// TIA Portal V18 export
PlcTagTable "Default tag table"
  PlcTag "HMI_Run_Enable"  LogicalAddress=%M20.0
  PlcTag "HMI_Reset_Alarm"  LogicalAddress=%M20.1
  PlcTag "HMI_Che_Do_Thi"  LogicalAddress=%M20.2
  PlcTag "HMI_Sim_Mode"  LogicalAddress=%M20.3
  PlcTag "PLC1_State"  LogicalAddress=%MW12
  PlcTag "PLC1_Loi_Tong"  LogicalAddress=%M20.4
  PlcTag "PLC1_Stop_Active"  LogicalAddress=%M20.5
  PlcTag "PLC1_EStop_Latch"  LogicalAddress=%M20.6
  PlcTag "PLC1_SP_Valid"  LogicalAddress=%M20.7
  PlcTag "Nut_Khoi_Dong_HMI"  LogicalAddress=%M21.0
  PlcTag "Nut_Dung_HMI"  LogicalAddress=%M21.1
  PlcTag "Nut_Reset_HMI"  LogicalAddress=%M21.2
  PlcTag "HMI_VFD_Bon2_Comm_Enable"  LogicalAddress=%M21.3
  PlcTag "HMI_VFD_Bon2_Real_Enable"  LogicalAddress=%M21.4
  PlcTag "HMI_PID_Bon2_Dau_Noi_Enable"  LogicalAddress=%M21.5
  PlcTag "PID_Bon2_Enable"  LogicalAddress=%M21.6
  PlcTag "PID_Bon2_Enable_Eff"  LogicalAddress=%M21.7
  PlcTag "PID_Bon2_SP"  LogicalAddress=%MD30
  PlcTag "PID_Bon2_PV_Eff"  LogicalAddress=%MD34
  PlcTag "PID_Bon2_CV"  LogicalAddress=%MD38
  PlcTag "HMI_SP_PLC1_Nhiet_Do_Bon2"  LogicalAddress=%MD42
  PlcTag "HMI_SP_PLC1_Toc_Do_Bon2_Main"  LogicalAddress=%MD46
  PlcTag "TT3208_Bon2_Eff"  LogicalAddress=%MD50
  PlcTag "TT3208_Bon2_HMI"  LogicalAddress=%MD54
  PlcTag "VFD_Bon2_Toc_Do_Cmd"  LogicalAddress=%MD58
  PlcTag "TT3208_Bon2_Use_HMI"  LogicalAddress=%M22.0
  PlcTag "VFD_Bon2_MB_Error"  LogicalAddress=%M22.1
  PlcTag "VFD_Bon2_MB_Busy"  LogicalAddress=%M22.2
  PlcTag "VFD_Bon2_MB_Done"  LogicalAddress=%M22.3
  PlcTag "MB_TCP_ERROR"  LogicalAddress=%M22.4
  PlcTag "MB_TCP_BUSY"  LogicalAddress=%M22.5
  PlcTag "MB_TCP_DONE"  LogicalAddress=%M22.6
  PlcTag "PLC1_Heartbeat_Timeout"  LogicalAddress=%M22.7
  PlcTag "VFD_Bon2_MB_ControlWord"  LogicalAddress=%MW62
  PlcTag "VFD_Bon2_MB_StatusWord"  LogicalAddress=%MW64
  PlcTag "VFD_Bon2_MB_FreqSetpoint"  LogicalAddress=%MW66
  PlcTag "VFD_Bon2_MB_FreqActual"  LogicalAddress=%MW68
  PlcTag "VFD_Bon2_MB_Status"  LogicalAddress=%MW70
  PlcTag "MB_TCP_STATUS"  LogicalAddress=%MW72
  PlcTag "MB_TCP_iStep"  LogicalAddress=%MW74
  PlcTag "PLC1_Heartbeat"  LogicalAddress=%MW76
  PlcTag "PLC2_Heartbeat_Recv"  LogicalAddress=%MW78
  PlcTag "VFD_Bon2_Contactor"  LogicalAddress=%Q0.0
  PlcTag "CV3201_Nuoc_Bon1_M"  LogicalAddress=%MD1200
  PlcTag "CV3206_Hoi_Bon2_M"  LogicalAddress=%MD1208
  PlcTag "CV3304_Nuoc_Lam_Mat_M"  LogicalAddress=%MD1232
  PlcTag "FQ3200_Bon1_Eff"  LogicalAddress=%MD712
  PlcTag "FQ3205_Bon2_Eff"  LogicalAddress=%MD744
  PlcTag "FT3309_Xa_Thanh_Pham_Eff"  LogicalAddress=%MD880
  PlcTag "HMI_Anim_Bon1_Frame"  LogicalAddress=%MW260
  PlcTag "HMI_Anim_Bon1_MucDich"  LogicalAddress=%MW262
  PlcTag "HMI_Anim_Bon2_Frame"  LogicalAddress=%MW264
  PlcTag "HMI_Anim_Bon2_MucDich"  LogicalAddress=%MW266
  PlcTag "HMI_Anim_BonChua1_MucDich"  LogicalAddress=%MW268
  PlcTag "HMI_Anim_BonChua2_MucDich"  LogicalAddress=%MW270
  PlcTag "LT3203_Bon1_Eff"  LogicalAddress=%MD720
  PlcTag "LT3209_Bon2_Eff"  LogicalAddress=%MD752
  PlcTag "LT3302_BonChua1_Eff"  LogicalAddress=%MD832
  PlcTag "LT3307_BonChua2_Eff"  LogicalAddress=%MD856
  PlcTag "PI3308_Truoc_Filter_Eff"  LogicalAddress=%MD872
  PlcTag "Pump3264_Chuyen_Nhanh1"  LogicalAddress=%M100.0
  PlcTag "Pump3265_Chuyen_Nhanh2"  LogicalAddress=%M100.1
  PlcTag "Pump3361_LuanChuyen_BonChua1"  LogicalAddress=%M100.2
  PlcTag "Pump3362_Xa_BonChua1"  LogicalAddress=%M100.3
  PlcTag "Pump3364_Filter"  LogicalAddress=%M100.4
  PlcTag "Pump3365_Filter"  LogicalAddress=%M100.5
  PlcTag "TT3204_Bon1_Eff"  LogicalAddress=%MD728
  PlcTag "TT3301_BonChua1_Eff"  LogicalAddress=%MD840
  PlcTag "TT3303_TraoDoiNhiet_Eff"  LogicalAddress=%MD848
  PlcTag "TT3306_BonChua2_Eff"  LogicalAddress=%MD864
  PlcTag "V3230_Nuoc_Bon1"  LogicalAddress=%M100.6
  PlcTag "V3232_Xa_Bon1"  LogicalAddress=%M100.7
  PlcTag "V3233_Xa_Bon1"  LogicalAddress=%M101.0
  PlcTag "V3234_Xa_Bon1"  LogicalAddress=%M101.1
  PlcTag "V3235_Nuoc_Bon2"  LogicalAddress=%M101.2
  PlcTag "V3237_Xa_Bon2"  LogicalAddress=%M101.3
  PlcTag "V3238_Xa_Bon2"  LogicalAddress=%M101.4
  PlcTag "V3239_Xa_Bon2"  LogicalAddress=%M101.5
  PlcTag "V3331_Xa_BonChua1"  LogicalAddress=%M101.6
  PlcTag "V3332_Xa_BonChua1"  LogicalAddress=%M101.7
  PlcTag "V3333_DieuHuong_BonChua1"  LogicalAddress=%M102.0
  PlcTag "V3334_DieuHuong_BonChua1"  LogicalAddress=%M102.1
  PlcTag "V3335_DieuHuong_BonChua1"  LogicalAddress=%M102.2
  PlcTag "V3338_Xa_BonChua2"  LogicalAddress=%M102.3
  PlcTag "V3339_Xa_BonChua2"  LogicalAddress=%M102.4
  PlcTag "V3340_Duong_Filter"  LogicalAddress=%M102.5
  PlcTag "V3341_Duong_Filter"  LogicalAddress=%M102.6
  PlcTag "HMI_SP_PLC1_Nuoc_Bon1"  LogicalAddress=%MD896
  PlcTag "HMI_SP_PLC1_Nuoc_Bon2"  LogicalAddress=%MD900
  PlcTag "HMI_SP_Time_Khuay_Bon1"  LogicalAddress=%MD944
  PlcTag "HMI_SP_Time_Fwd"  LogicalAddress=%MD952
  PlcTag "HMI_SP_Time_Rev"  LogicalAddress=%MD956
  PlcTag "HMI_SP_Time_Sterilize"  LogicalAddress=%MD960
